{attribute 'qualified_only'}
{attribute 'strict'}
{attribute 'to_string'}
TYPE E_Warn :
(
	Warn000,
	Warn001,
	Warn002,
	Warn003,
	Warn004,
	Warn005,
	Warn006,
	Warn007,
	Warn008,
	Warn009,
	Warn010,
	Warn011,
	Warn012,
	Warn013,
	Warn014,
	Warn015,
	Warn016,
	Warn017,
	Warn018,
	Warn019,
	Warn020,
	Warn021,
	Warn022,
	Warn023,
	Warn024,
	Warn025,
	Warn026,
	Warn027,
	Warn028,
	Warn029,
	Warn030,
	Warn031,
	Warn032,
	Warn033,
	Warn034,
	Warn035,
	Warn036,
	Warn037,
	Warn038,
	Warn039,
	Warn040,
	Warn041,
	Warn042,
	Warn043,
	Warn044,
	Warn045,
	Warn046,
	Warn047,
	Warn048,
	Warn049,
	Warn050,
	Warn051,
	Warn052,
	Warn053,
	Warn054,
	Warn055,
	Warn056,
	Warn057,
	Warn058,
	Warn059,
	Warn060,
	Warn061,
	Warn062,
	Warn063,
	Warn064,
	Warn065,
	Warn066,
	Warn067,
	Warn068,
	Warn069,
	Warn070,
	Warn071,
	Warn072,
	Warn073,
	Warn074,
	Warn075,
	Warn076,
	Warn077,
	Warn078,
	Warn079,
	Warn080,
	Warn081,
	Warn082,
	Warn083,
	Warn084,
	Warn085,
	Warn086,
	Warn087,
	Warn088,
	Warn089,
	Warn090,
	Warn091,
	Warn092,
	Warn093,
	Warn094,
	Warn095,
	Warn096,
	Warn097,
	Warn098,
	Warn099,
	Warn100,
	Warn101,
	Warn102,
	Warn103,
	Warn104,
	Warn105,
	Warn106,
	Warn107,
	Warn108,
	Warn109,
	Warn110,
	Warn111,
	Warn112,
	Warn113,
	Warn114,
	Warn115,
	Warn116,
	Warn117,
	Warn118,
	Warn119,
	Warn120,
	Warn121,
	Warn122,
	Warn123,
	Warn124,
	Warn125,
	Warn126,
	Warn127,
	Warn128,
	Warn129,
	Warn130,
	Warn131,
	Warn132,
	Warn133,
	Warn134,
	Warn135,
	Warn136,
	Warn137,
	Warn138,
	Warn139,
	Warn140,
	Warn141,
	Warn142,
	Warn143,
	Warn144,
	Warn145,
	Warn146,
	Warn147,
	Warn148,
	Warn149,
	Warn150,
	Warn151,
	Warn152,
	Warn153,
	Warn154,
	Warn155,
	Warn156,
	Warn157,
	Warn158,
	Warn159,
	Warn160,
	Warn161,
	Warn162,
	Warn163,
	Warn164,
	Warn165,
	Warn166,
	Warn167,
	Warn168,
	Warn169,
	Warn170,
	Warn171,
	Warn172,
	Warn173,
	Warn174,
	Warn175,
	Warn176,
	Warn177,
	Warn178,
	Warn179,
	Warn180,
	Warn181,
	Warn182,
	Warn183,
	Warn184,
	Warn185,
	Warn186,
	Warn187,
	Warn188,
	Warn189,
	Warn190,
	Warn191,
	Warn192,
	Warn193,
	Warn194,
	Warn195,
	Warn196,
	Warn197,
	Warn198,
	Warn199,
	Warn200,
	Warn201,
	Warn202,
	Warn203,
	Warn204,
	Warn205,
	Warn206,
	Warn207,
	Warn208,
	Warn209,
	Warn210,
	Warn211,
	Warn212,
	Warn213,
	Warn214,
	Warn215,
	Warn216,
	Warn217,
	Warn218,
	Warn219,
	Warn220,
	Warn221,
	Warn222,
	Warn223,
	Warn224,
	Warn225,
	Warn226,
	Warn227,
	Warn228,
	Warn229,
	Warn230,
	Warn231,
	Warn232,
	Warn233,
	Warn234,
	Warn235,
	Warn236,
	Warn237,
	Warn238,
	Warn239,
	Warn240,
	Warn241,
	Warn242,
	Warn243,
	Warn244,
	Warn245,
	Warn246,
	Warn247,
	Warn248,
	Warn249,
	Warn250,
	Warn251,
	Warn252,
	Warn253,
	Warn254,
	Warn255,
	Warn256,
	Warn257,
	Warn258,
	Warn259,
	Warn260,
	Warn261,
	Warn262,
	Warn263,
	Warn264,
	Warn265,
	Warn266,
	Warn267,
	Warn268,
	Warn269,
	Warn270,
	Warn271,
	Warn272,
	Warn273,
	Warn274,
	Warn275,
	Warn276,
	Warn277,
	Warn278,
	Warn279,
	Warn280,
	Warn281,
	Warn282,
	Warn283,
	Warn284,
	Warn285,
	Warn286,
	Warn287,
	Warn288,
	Warn289,
	Warn290,
	Warn291,
	Warn292,
	Warn293,
	Warn294,
	Warn295,
	Warn296,
	Warn297,
	Warn298,
	Warn299,
	Warn300,
	Warn301,
	Warn302,
	Warn303,
	Warn304,
	Warn305,
	Warn306,
	Warn307,
	Warn308,
	Warn309,
	Warn310,
	Warn311,
	Warn312,
	Warn313,
	Warn314,
	Warn315,
	Warn316,
	Warn317,
	Warn318,
	Warn319,
	Warn320,
	Warn321,
	Warn322,
	Warn323,
	Warn324,
	Warn325,
	Warn326,
	Warn327,
	Warn328,
	Warn329,
	Warn330,
	Warn331,
	Warn332,
	Warn333,
	Warn334,
	Warn335,
	Warn336,
	Warn337,
	Warn338,
	Warn339,
	Warn340,
	Warn341,
	Warn342,
	Warn343,
	Warn344,
	Warn345,
	Warn346,
	Warn347,
	Warn348,
	Warn349,
	Warn350,
	Warn351,
	Warn352,
	Warn353,
	Warn354,
	Warn355,
	Warn356,
	Warn357,
	Warn358,
	Warn359,
	Warn360,
	Warn361,
	Warn362,
	Warn363,
	Warn364,
	Warn365,
	Warn366,
	Warn367,
	Warn368,
	Warn369,
	Warn370,
	Warn371,
	Warn372,
	Warn373,
	Warn374,
	Warn375,
	Warn376,
	Warn377,
	Warn378,
	Warn379,
	Warn380,
	Warn381,
	Warn382,  
	Warn383,
	Warn384,
	Warn385,
	Warn386,
	Warn387,
	Warn388,
	Warn389,  
	Warn390,
	Warn391,
	Warn392,
	Warn393,
	Warn394,
	Warn395,
	Warn396,
	Warn397,
	Warn398,
	Warn399,
	Warn400,//B槽主軸伺服馬達_驅動器異常   
	Warn401,//B槽清洗內罩升降1馬達_驅動器異常
	Warn402,//B槽清洗內罩升降2馬達_驅動器異常
	Warn403,//B槽清洗外罩升降1馬達_驅動器異常
	Warn404,//B槽清洗外罩升降2馬達_驅動器異常
	Warn405,//B槽噴頭擺臂升降馬達_驅動器異常 
	Warn406,//B槽噴頭擺臂馬達_驅動器異常   
	Warn407,//B槽頂PIN升降馬達_驅動器異常 
	Warn408,//B槽噴頭X軸馬達_驅動器異常   
	Warn409,//B槽噴頭Y1軸馬達_驅動器異常  
	Warn410,//B槽噴頭Y2軸馬達_驅動器異常  
	Warn411,//B槽噴頭Z軸馬達_驅動器異常   
	Warn412,//B槽噴頭T軸馬達_驅動器異常   
	Warn413,//
	Warn414,//
	Warn415,//
	Warn416,//
	Warn417,//
	Warn418,//
	Warn419,//
	Warn420,//
	Warn421,//
	Warn422,//
	Warn423,//
	Warn424,//
	Warn425,//
	Warn426,//
	Warn427,//
	Warn428,//
	Warn429,//
	Warn430,//
	Warn431,//
	Warn432,//
	Warn433,//
	Warn434,//
	Warn435,//
	Warn436,//
	Warn437,//
	Warn438,//
	Warn439,//
	Warn440,//
	Warn441,//
	Warn442,//
	Warn443,//
	Warn444,//
	Warn445,//
	Warn446,//
	Warn447,//
	Warn448,//
	Warn449,//
	Warn450,//
	Warn451,//
	Warn452,//
	Warn453,//
	Warn454,//
	Warn455,//
	Warn456,//
	Warn457,//                 
	Warn458,//                 
	Warn459,//                 
	Warn460,//                 
	Warn461,//                 
	Warn462,//                 
	Warn463,//                 
	Warn464,//                 
	Warn465,//                 
	Warn466,//                 
	Warn467,//                 
	Warn468,//                 
	Warn469,//                 
	Warn470,//                 
	Warn471,//                 
	Warn472,//                 
	Warn473,//                 
	Warn474,//                 
	Warn475,//                 
	Warn476,//                 
	Warn477,//                 
	Warn478,//                 
	Warn479,//                 
	Warn480,//                 
	Warn481,//                 
	Warn482,//                 
	Warn483,//                 
	Warn484,//                 
	Warn485,//                 
	Warn486,//                 
	Warn487,//                 
	Warn488,//                 
	Warn489,//                 
	Warn490,//                 
	Warn491,//                 
	Warn492,//                 
	Warn493,//                 
	Warn494,//                 
	Warn495,//                 
	Warn496,//                 
	Warn497,//                 
	Warn498,//                 
	Warn499,//                 
	Warn500,//                 
	Warn501,//                 
	Warn502,//                 
	Warn503,//                 
	Warn504,//                 
	Warn505,//                 
	Warn506,//                 
	Warn507,//                 
	Warn508,//                 
	Warn509,//                 
	Warn510,//                 
	Warn511,//                 
	Warn512,//                 
	Warn513,//                 
	Warn514,//                 
	Warn515,//                 
	Warn516,//                 
	Warn517,//                 
	Warn518,//                 
	Warn519,//                 
	Warn520,//                 
	Warn521,//                 
	Warn522,//                 
	Warn523,//                 
	Warn524,//                 
	Warn525,//                 
	Warn526,//                 
	Warn527,//                 
	Warn528,//                 
	Warn529,//                 
	Warn530,//                 
	Warn531,//                 
	Warn532,//                 
	Warn533,//                 
	Warn534,//                 
	Warn535,//                 
	Warn536,//                 
	Warn537,//                 
	Warn538,//                 
	Warn539,//                 
	Warn540,//                 
	Warn541,//                 
	Warn542,//                 
	Warn543,//                 
	Warn544,//                 
	Warn545,//                 
	Warn546,//                 
	Warn547,//                 
	Warn548,//                 
	Warn549,//                 
	Warn550,//                 
	Warn551,//                 
	Warn552,//                 
	Warn553,//                 
	Warn554,//                 
	Warn555,//                 
	Warn556,//                 
	Warn557,//                 
	Warn558,//                 
	Warn559,//                 
	Warn560,//                 
	Warn561,//                 
	Warn562,//                 
	Warn563,//                 
	Warn564,//                 
	Warn565,//                 
	Warn566,//                 
	Warn567,//                 
	Warn568,//                 
	Warn569,//                 
	Warn570,//                 
	Warn571,//                 
	Warn572,//                 
	Warn573,//                 
	Warn574,//                 
	Warn575,//                 
	Warn576,//                 
	Warn577,//                 
	Warn578,//                 
	Warn579,//                 
	Warn580,//                 
	Warn581,//                 
	Warn582,//                 
	Warn583,//                 
	Warn584,//                 
	Warn585,//                 
	Warn586,//                 
	Warn587,//                 
	Warn588,//                 
	Warn589,//                 
	Warn590,//                 
	Warn591,//                 
	Warn592,//                 
	Warn593,//                 
	Warn594,//                 
	Warn595,//                 
	Warn596,//                 
	Warn597,//                 
	Warn598,//                 
	Warn599 //                 
);
END_TYPE

(* stored: Version 1.1.0.1, ProductVersion 3.1.4026.18
   DUT E_Warn: Id {07a88125-4f96-4f66-96dc-8a283f5f706f} *)
